(* PLC project output_chain_control, Dassault Systèmes ControlBuild 2024x *)
(* stored: creationDateTime 2023-10-03T11:13:58-01:00 *)

FUNCTION_BLOCK tri_chain.output_chain_control
  VAR_INPUT
    globalRunning : BOOL := false;
    depositEnabled : BOOL := false;
    endSensor : BOOL := false;
  END_VAR
  VAR_OUTPUT
    movement : BOOL := false;
  END_VAR

INITIAL_STEP 10:
  COMPUTE_FUNCTION_BLOCKS(S);
END_STEP
TRANSITION FROM 10 TO 11
  := depositEnabled AND globalRunning;
END_TRANSITION
STEP 11:
  11_INLINE1(N);
END_STEP
ACTION 11_INLINE1:
  movement;
END_ACTION
TRANSITION FROM 11 TO 12
  := endSensor;
END_TRANSITION
STEP 12:
  12_INLINE2(N);
END_STEP
ACTION 12_INLINE2:
  movement;
END_ACTION
TRANSITION FROM 12 TO 10
  := NOT endSensor;
END_TRANSITION
ACTION COMPUTE_FUNCTION_BLOCKS:  (* blocks drawn on the SFC sheet *)
  G1:
END_ACTION
END_FUNCTION_BLOCK
